(* PLC project Unnamed, Unknown Unnamed 1 *)
(* stored: creationDateTime 2026-03-03T09:36:26, modificationDateTime 2026-03-03T09:50:58 *)

PROGRAM program0
  VAR
    JOG_PB_RAW AT %IX0.6 : BOOL;
    JOG_PB_VALID AT %M0.4 : BOOL;
  END_VAR
  VAR
    TON0 : TON;
  END_VAR

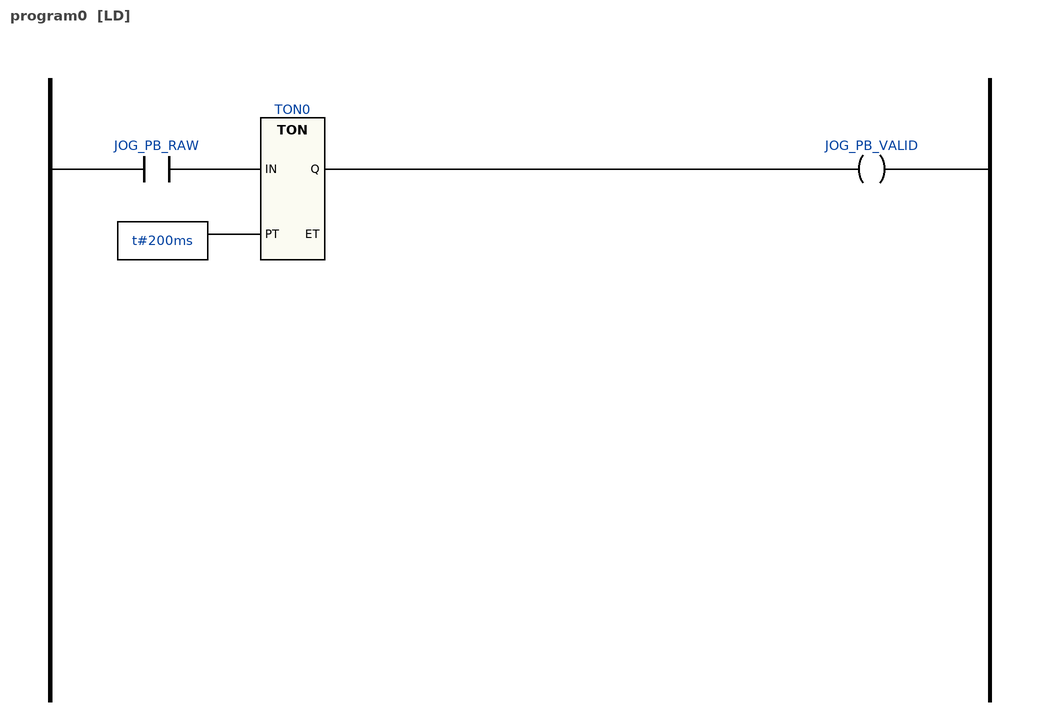
(* LD diagram, written out as Structured Text *)
TON0(IN := JOG_PB_RAW, PT := t#200ms);
JOG_PB_VALID := TON0.Q;
END_PROGRAM

CONFIGURATION Config0
  RESOURCE Res0 ON PLC
    TASK task0(INTERVAL := T#20ms, PRIORITY := 0);
    PROGRAM instance0 WITH task0 : program0;
  END_RESOURCE
END_CONFIGURATION
